// TIA Portal V20 export
DATA_BLOCK "T1-A ARUNC I-O"   // DB1602
{ S7_Optimized_Access := 'TRUE' }
AUTHOR : SAS
// stored: AutoNumber false, IsRetainMemResEnabled true, MemoryReserve 100, RetainMemoryReserve 100
   VAR
      DI : Struct
         "F8.1" : Bool;   // (E25.0) T1A Prezenta Tensiune Alimentare ElectroValva Arunctor
         "S44.6" : Bool;   // (E25.7) T1A Aruncator Comanda ''Ridicare''
         "S44.7" : Bool;   // (E26.0) T1A Aruncator Comanda 'Coborare'
         "S44.8" : Bool;   // (E26.7) T1A-Aruncator: Scuturator
         "B48.1" : Bool;   // (E30.0) T1A Aruncator Senzor Prozimitate Pozitia 'Jos'
         "B48.2" : Bool;   // (E30.1) T1A Aruncator Senzor Prozimitate Pozitia 'Sus'
      END_STRUCT;
      "DO" : Struct
         "K56.1" : Bool;   // (A24.0) T1A Aruncator ElectroValva ''Ridicare''
         "A24.3" : Bool;   // (A24.3) Comanda scuturator T1A
      END_STRUCT;
   END_VAR
BEGIN
END_DATA_BLOCK
